Fanuc KAREL source: f_attr2_t.kl

PROGRAM F_ATTR2_T
%LOCKGROUP = 1
%NOSCANSVARS
%SHADOWVARS
%CMOS2SHADOW
%FLASHROM
%POWERFAIL
%RWACCESS
VAR
  i : INTEGER
BEGIN
  i = 1
END F_ATTR2_T
